RoboDK station: UR5 Tufting.rdk

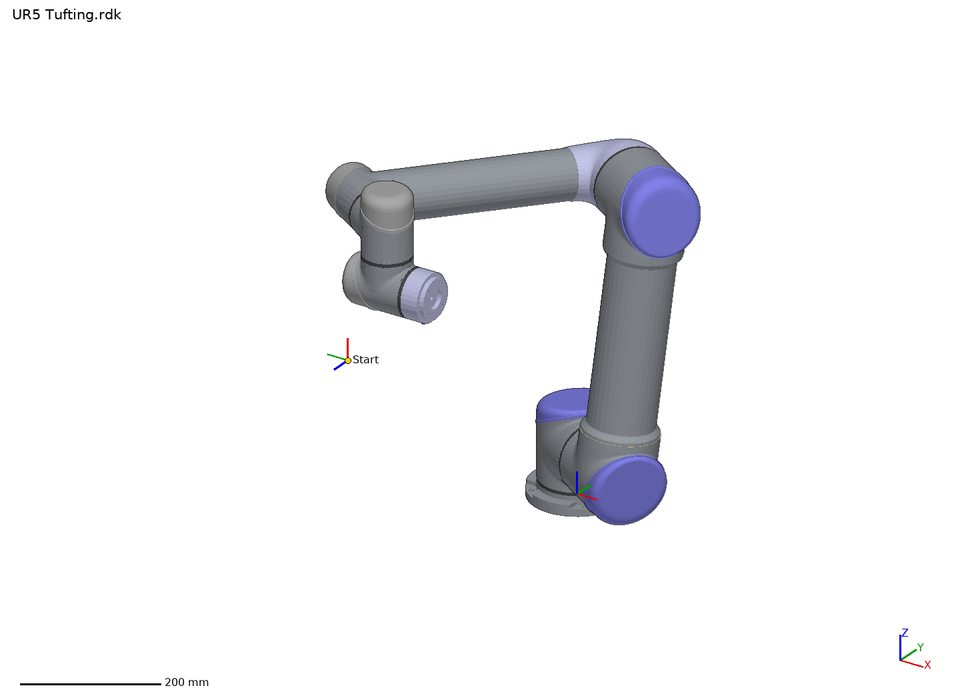
[picture v0: the station drawn from its stored meshes, robots at their saved joint values, targets as dots, program paths as lines]
Station UR5 Tufting. Poses are relative to the parent item; angles as X-Y-Z fixed-axis rotations.
  - frame UR5 Base at (0, 0, 0) mm
    - robot UR5: 6 axes, payload 5 kg, reach 850 mm, repeatability 0.1 mm, weight 18.4 kg
        modified DH rows (alpha deg, a mm, theta deg, d mm): 0, 0, 0, 89.2; 90, 0, 180, 0; 0, 425, 0, 0; 0, 392.43, 0, 109; -90, 0, 0, 93.65; 90, 0, 180, 82
        joint limits [-360, -360, -360, -360, -360, -360] to [360, 360, 360, 360, 360, 360]; home [0, -90, -90, 0, 90, 0]; saved at [57.801, -97.212, 93.681, 3.529, -33.712, 0.001]
      - tool Tool, TCP at (-188.9, 3.33, 9.46) mm, rotated rx -90 ry 0 rz 90 deg
    - frame Canvas at (9.55, -580.81, 444.73) mm, rotated rx 0 ry -90 rz 91.5 deg
      - target Start (Cartesian target) at (0, 0, 0) mm; joints [81.092, -70.487, 69.49, 21.352, -10.582, -19.072] of UR5
